{attribute 'hide_all_locals'}
FUNCTION_BLOCK FB_SPOpt_HybridAirSystem
VAR_INPUT PERSISTENT
	bEnable							: BOOL;									//Enable or dissable thsi Function
END_VAR
VAR_INPUT
	byStateSystemIn					: BYTE;									//Actual State from the System. 0 = off, 1 = Heating mode on, 2 = Cooling Mode on
	rFlowAirTempIn					: REAL;									//Actual Flow Air Temperature
	rReturnAirTempIn				: REAL;									//Actual Return Air Temperature
	rInToOutAirTempIn				: REAL;									//Actual outdoor air flow temperature
	rOutToInAirTempIn				: REAL;									//Actual indoor air flow temperature
END_VAR
VAR_OUTPUT
	bError							: BOOL;									//Error from this Fuction
	byStateSystemOut				: BYTE;									//{#lynus.ag#()} //State from the System. 0 = off, 1 = Heating mode on, 2 = Cooling Mode on		
	rFlowAirTempOut					: REAL;									//{#lynus.ag#()} //Flow Air Temperature to send to the Backend Service.
	rReturnAirTempOut				: REAL;									//{#lynus.ag#()} //Return Air Temperature to send to the Backend Service.
	rInToOutAirTempOut				: REAL;									//{#lynus.ag#()} //Outdoor air flow temperature to send to the Backend Service.
	rOutToInAirTempOut				: REAL;									//{#lynus.ag#()} //Indoor air flow temperature to send to the Backend Service.
	diNrOfSPOpt_OUT					: DINT;									//Active Number from Setpoint Optimizer for using on other functions
END_VAR
VAR
	fbNumberDevice					: FB_NumberOfDevice;					//Function block to calcualte the number of the Device
	timDissableFunctions			: TON;									//Timer to dissable the Function after Lynus_Standards.Constants_General.tTimeDissableLynusFunctions Days without connection to the Lynus Cloud
	timResetConnectionOnGVL			: TON;									//Timer to try reset the connection Flag on the GVL. (When somebody delete the Connection Function and make only a onlinechange)
END_VAR

//Creator : Kai Ebensperger
//Company : Lynus AG
//Date : 03.12.2021
//Version : 1.0.0.0

//This Function is a Help Function for the Setpoint Optimizer on our Backend System
//Here we can read in the neccessary Values for a Hybrid Air System from a external Service and can send then to the Backend System for optimizing
//Hybrid System can bee heating and cooling
//Its Helpfull if we work with the TMC File

(*----------------------------------------------------------------------------------------Limits---------------------------------------------------------------------------------------------------------------*)

byStateSystemIn := LIMIT(0,byStateSystemIn,2);
	rFlowAirTempIn := LIMIT(-30,rFlowAirTempIn,150);
		rReturnAirTempIn := LIMIT(-30,rReturnAirTempIn,150);
			rInToOutAirTempIn := LIMIT(-30,rInToOutAirTempIn,150);
				rOutToInAirTempIn := LIMIT(-30,rOutToInAirTempIn,150);

(*-------------------------------------------------------------Calcualte the number of SP Opttimizer---------------------------------------------------------------*)

fbNumberDevice(
	diActualNumberOfDevices:= Lynus_Standards.GVL_Energy.stNumberOfDevices.diNumberOfSetPointOpt, 
	diMaxNumberOfDevices:= Constants_Energy.diMaxNumberOfSetPointOpt, 
	udiCounterOnlineChange:= TwinCAT_SystemInfoVarList._AppInfo.OnlineChangeCnt, 
	bNumberIsCalculatet=> , 
	bFPNumberIsCalculatet=> , 
	bOnlineChange=> , 
	diNumberForThisDevice=> diNrOfSPOpt_OUT, 
	diNumberOfTotalDevices=> );

//Write new Numer on GVL
IF fbNumberDevice.bFPNumberIsCalculatet THEN
	Lynus_Standards.GVL_Energy.stNumberOfDevices.diNumberOfSetPointOpt := fbNumberDevice.diNumberOfTotalDevices;	
END_IF 

//Delete old Number on GVL
IF fbNumberDevice.bOnlineChange THEN 
	Lynus_Standards.GVL_Energy.stNumberOfDevices.diNumberOfSetPointOpt := diNrOfSPOpt_OUT;
END_IF								
				
(*-------------------------------------------------------------Service from Backend is ready and check the connection to backen for dissabel/enable EMS Function---------------------------------------------------------------*)

//Try to reset the variable for connection on the GVL. When all is normal then the Lynus Mqtt connection function set this variable to true in the next cycle
//When we have no connection to the backend or no HB from the Service then after Lynus_Standards.Constants_General.tTimeDissableLynusFunctions days the EMS is dissabled with all of his functionalities
timResetConnectionOnGVL(IN:= NOT timResetConnectionOnGVL.Q, PT:= T#1H, Q=> , ET=> );
	IF timResetConnectionOnGVL.Q THEN Lynus_Standards.GVL_Communicator.bStateConnectionToEnableFunctions := FALSE; END_IF
		IF NOT Lynus_Standards.GVL_Communicator.bStateConnectionToEnableFunctions THEN timDissableFunctions.IN := TRUE; ELSE timDissableFunctions.IN := FALSE; END_IF  
			timDissableFunctions(IN:= , PT:= Lynus_Standards.Constants_General.tTimeDissableLynusFunctions, Q=> , ET=> );

(*------------------------------------------------------------------Error----------------------------------------------------------------------------*)	

IF Lynus_Standards.GVL_Energy.stNumberOfDevices.diNumberOfSetPointOpt > Constants_Energy.diMaxNumberOfSetPointOpt THEN bError := TRUE; ELSE bError := FALSE; END_IF 			
			
(*-------------------------------------------------------------------------------------In to Out---------------------------------------------------------------------------------------*)

byStateSystemOut := byStateSystemIn;
	rFlowAirTempOut := rFlowAirTempIn;
		rReturnAirTempOut := rReturnAirTempIn;	
			rInToOutAirTempOut := rInToOutAirTempIn;
				rOutToInAirTempOut := rOutToInAirTempIn;		

IF NOT bEnable OR timDissableFunctions.Q OR Lynus_Standards.GVL_Energy.stNumberOfDevices.diNumberOfSetPointOpt > Constants_Energy.diMaxNumberOfSetPointOpt THEN
	byStateSystemOut := 0;	
END_IF

END_FUNCTION_BLOCK

(* stored: Version 1.1.0.1, ProductVersion 3.1.4024.9
   POU FB_SPOpt_HybridAirSystem: Id {36f0f71d-428b-4343-ade8-73d05db32f99}, SpecialFunc None *)
